// Mitsubishi GX Works2 project: PLC_GROUP18   PLC: FX3G
// פרויקט אוטומציה

// global labels: Global1
VAR_GLOBAL
  StartWorkingDay AT X007 : BOOL;
  EmergencyButton AT X005 : BOOL;
  WorkingDay AT Y007 : BOOL;
  InputChocolate AT D1101 : REAL;
  InputNuts AT D1103 : REAL;
  InputPistacho AT D1105 : REAL;
  InputKadaif AT D1107 : REAL;
  M_20 AT M20 : BOOL;
END_VAR
VAR_GLOBAL CONSTANT
  MinChocolate : REAL := 400.0;
  MinNuts : REAL := 100.0;
  MinPistacho : REAL := 120.0;
  MinKadaif : REAL := 60.0;
END_VAR
VAR_GLOBAL
  StockChocolate AT D1109 : REAL;
  StockNuts AT D1111 : REAL;
  StockPistacho AT D1113 : REAL;
  StockKadaif AT D1115 : REAL;
  M_21 AT M21 : BOOL;
  StartMelt AT X001 : BOOL;
  MeltContainer AT D1117 : REAL;
END_VAR
VAR_GLOBAL CONSTANT
  Choco_400 : REAL := 400.0;
END_VAR
VAR_GLOBAL
  MeltProcess AT Y001 : BOOL;
  CastingTime AT TC1 : BOOL;
END_VAR
VAR_GLOBAL CONSTANT
  DoneMelt : INT := 45;
END_VAR
VAR_GLOBAL
  FinishCasting AT TS1 : BOOL;
  SampleType AT X004 : BOOL;
  AnalogInput1 AT D8280 : INT;
  FloatInput1 AT D1119 : REAL;
  M_22 AT M22 : BOOL;
  M_23 AT M23 : BOOL;
  M_24 AT M24 : BOOL;
  M_25 AT M25 : BOOL;
END_VAR
VAR_GLOBAL CONSTANT
  Div400 : REAL := 400;
  Cons5 : REAL := 5.0;
END_VAR
VAR_GLOBAL
  MixNuts AT M26 : BOOL;
  DubalChoco AT M27 : BOOL;
END_VAR
VAR_GLOBAL CONSTANT
  Nuts100 : REAL := 100;
  Pistacho100 : REAL := 100;
END_VAR
VAR_GLOBAL
  FillContainer AT D1121 : REAL;
END_VAR
VAR_GLOBAL CONSTANT
  Amount200 : REAL := 200;
END_VAR
VAR_GLOBAL
  Sen_temp AT X002 : BOOL;
  EmplyTemplates AT X003 : BOOL;
END_VAR
VAR_GLOBAL CONSTANT
  Casting4sec : INT := 40;
END_VAR
VAR_GLOBAL
  CastingProcess AT Y002 : BOOL;
END_VAR
VAR_GLOBAL CONSTANT
  Nuts20 : REAL := 20;
  Pistacho120 : REAL := 120;
  Kadaif60 : REAL := 60;
END_VAR
VAR_GLOBAL
  Y_3 AT Y003 : BOOL;
  Y_4 AT Y004 : BOOL;
  TC_3 AT TC3 : BOOL;
END_VAR
VAR_GLOBAL CONSTANT
  FlashTime : INT := 10;
END_VAR
VAR_GLOBAL
  TS_3 AT TS3 : BOOL;
  TC_4 AT TC4 : BOOL;
  TS_4 AT TS4 : BOOL;
  Cooling AT X006 : BOOL;
END_VAR
VAR_GLOBAL CONSTANT
  Flash5 : INT := 50;
END_VAR
VAR_GLOBAL
  TC_2 AT TC2 : BOOL;
  TS_2 AT TS2 : BOOL;
  CoolContainer AT D1123 : REAL;
END_VAR
VAR_GLOBAL CONSTANT
  Cool3 : INT := 30;
END_VAR
VAR_GLOBAL
  CoolTime AT TC6 : BOOL;
  TS_6 AT TS6 : BOOL;
  CoolingProcess AT Y006 : BOOL;
  CastingContainer AT D1125 : REAL;
END_VAR
VAR_GLOBAL CONSTANT
  Reset : REAL;
END_VAR
VAR_GLOBAL
  M_28 AT M28 : BOOL;
  M_29 AT M29 : BOOL;
  X_0 AT X000 : BOOL;
  Y_5 AT Y005 : BOOL;
  FirstC AT CC1 : BOOL;
  OutC1 AT CS1 : BOOL;
END_VAR
VAR_GLOBAL CONSTANT
  CounterThreeTimes : WORD := 4;
END_VAR
VAR_GLOBAL
  FinishPacking AT M51 : BOOL;
  PacksContainer AT D1127 : REAL;
END_VAR
VAR_GLOBAL CONSTANT
  AddPack : REAL := 1;
END_VAR
VAR_GLOBAL
  M_52 AT M52 : BOOL;
  M_53 AT M53 : BOOL;
  M_60 AT M60 : BOOL;
  Packages AT D1129 : REAL;
  Analog_output AT D8282 : INT;
END_VAR
VAR_GLOBAL CONSTANT
  Cons40 : REAL := 40.0;
  ResetWord : INT;
END_VAR
VAR_GLOBAL
  X_10 AT X010 : BOOL;
  M_30 AT M30 : BOOL;
  M_31 AT M31 : BOOL;
END_VAR

// task Task_01 (event TRUE, interval 0, priority 31): POU_01

PROGRAM POU_01
(* structured ladder/FBD written out as ST: instructions are called as NAME(EN, inputs, outputs); _pN, _eN, _tN stand for wires *)
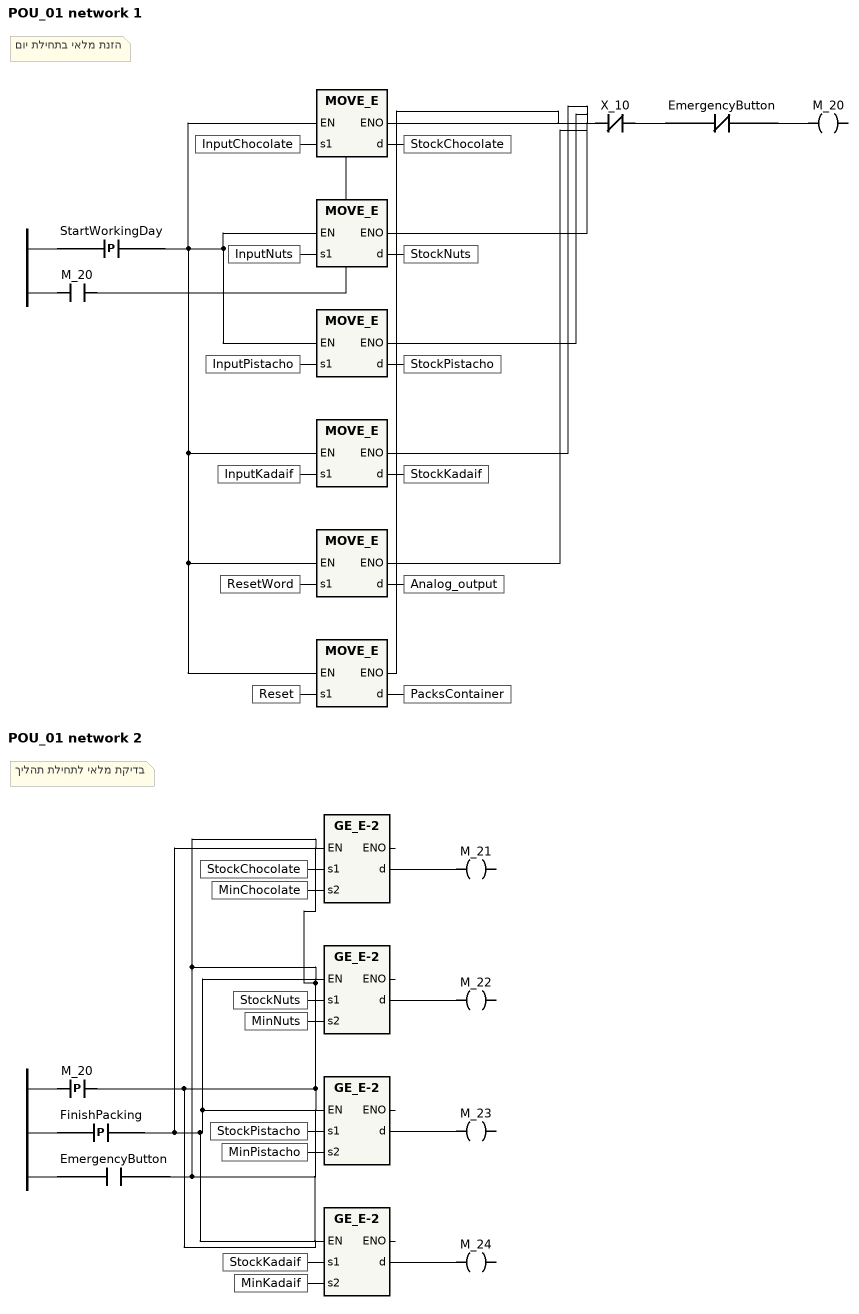
(* network 1 *)
(* הזנת מלאי בתחילת יום *)
_p1 := LDP(TRUE, StartWorkingDay);
_e2 := MOVE_E(_p1, InputChocolate, StockChocolate);
_e3 := MOVE_E(_p1, InputNuts, StockNuts);
_e4 := MOVE_E(_p1, InputPistacho, StockPistacho);
_e5 := MOVE_E(_p1, InputKadaif, StockKadaif);
_e6 := MOVE_E(_p1, ResetWord, Analog_output);
_e7 := MOVE_E(_p1, Reset, PacksContainer);
M_20 := ((_e2 OR _e3 OR _e4 OR _e5 OR _e6 OR _e7 OR M_20) AND NOT X_10) AND NOT EmergencyButton;
(* network 2 *)
(* בדיקת מלאי לתחילת תהליך *)
_p1 := LDP(TRUE, M_20) OR LDP(TRUE, FinishPacking) OR EmergencyButton;
GE_E(_p1, StockChocolate, MinChocolate, _t2);
M_21 := _t2;
GE_E(_p1, StockNuts, MinNuts, _t3);
M_22 := _t3;
GE_E(_p1, StockPistacho, MinPistacho, _t4);
M_23 := _t4;
GE_E(_p1, StockKadaif, MinKadaif, _t5);
M_24 := _t5;
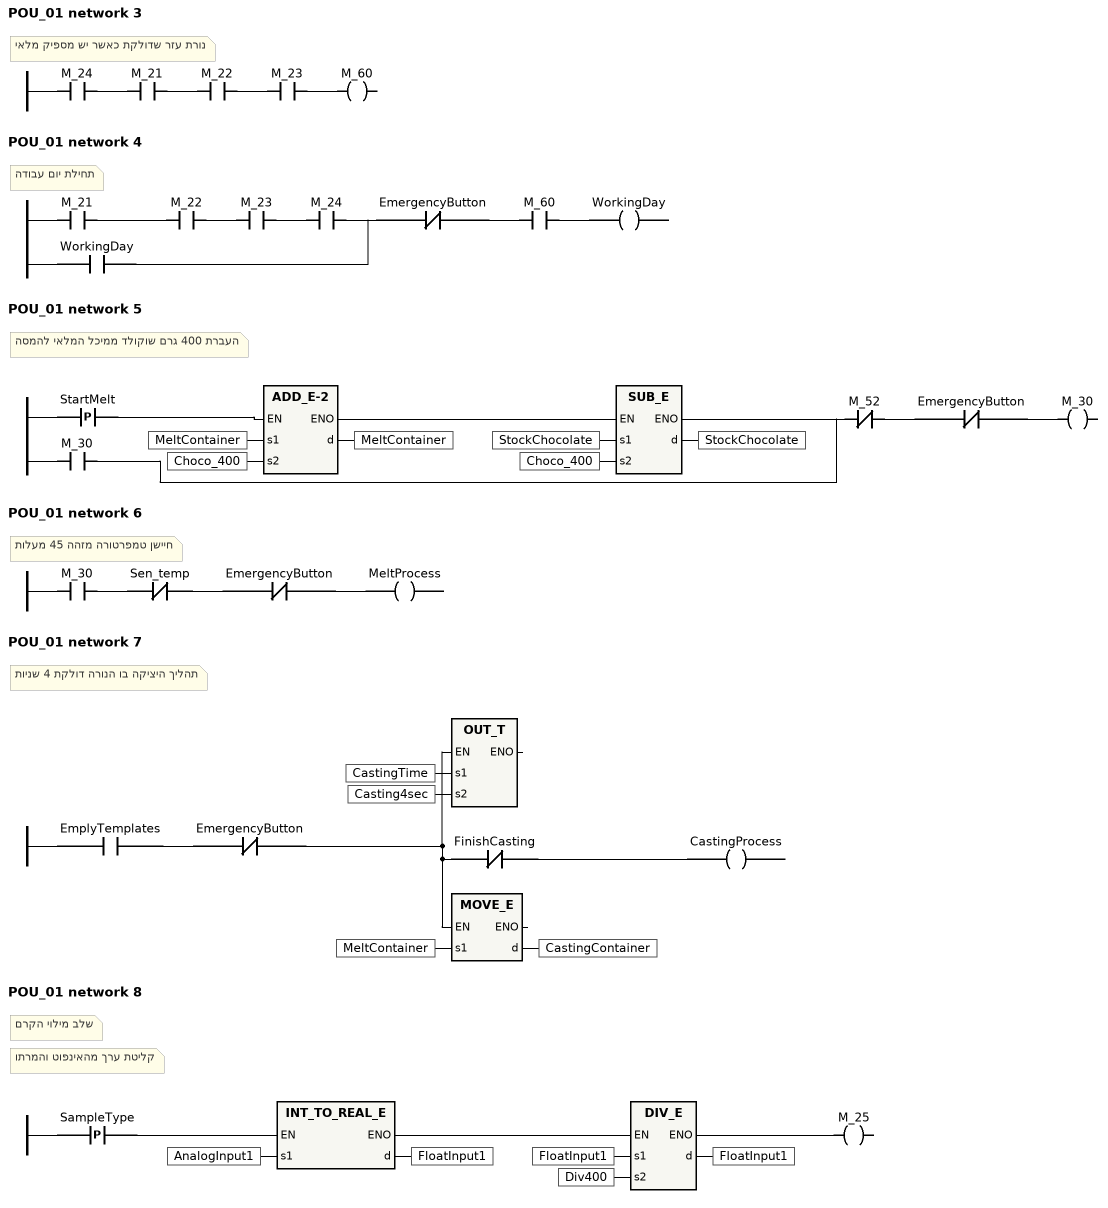
(* network 3 *)
(* נורת עזר שדולקת כאשר יש מספיק מלאי *)
M_60 := M_24 AND M_21 AND M_22 AND M_23;
(* network 4 *)
(* תחילת יום עבודה *)
WorkingDay := (((M_21 AND M_22 AND M_23 AND M_24) OR WorkingDay) AND NOT EmergencyButton) AND M_60;
(* network 5 *)
(* העברת 400 גרם שוקולד ממיכל המלאי להמסה *)
_e1 := ADD_E(LDP(TRUE, StartMelt), MeltContainer, Choco_400, MeltContainer);
_e2 := SUB_E(_e1, StockChocolate, Choco_400, StockChocolate);
M_30 := ((_e2 OR M_30) AND NOT M_52) AND NOT EmergencyButton;
(* network 6 *)
(* חיישן טמפרטורה מזהה 45 מעלות *)
MeltProcess := M_30 AND NOT Sen_temp AND NOT EmergencyButton;
(* network 7 *)
(* תהליך היציקה בו הנורה דולקת 4 שניות *)
_p1 := EmplyTemplates AND NOT EmergencyButton;
OUT_T(_p1, CastingTime, Casting4sec);
CastingProcess := _p1 AND NOT FinishCasting;
MOVE_E(_p1, MeltContainer, CastingContainer);
(* network 8 *)
(* שלב מילוי הקרם *)
(* קליטת ערך מהאינפוט והמרתו *)
_e1 := INT_TO_REAL_E(LDP(TRUE, SampleType), AnalogInput1, FloatInput1);
_e2 := DIV_E(_e1, FloatInput1, Div400, FloatInput1);
M_25 := _e2;
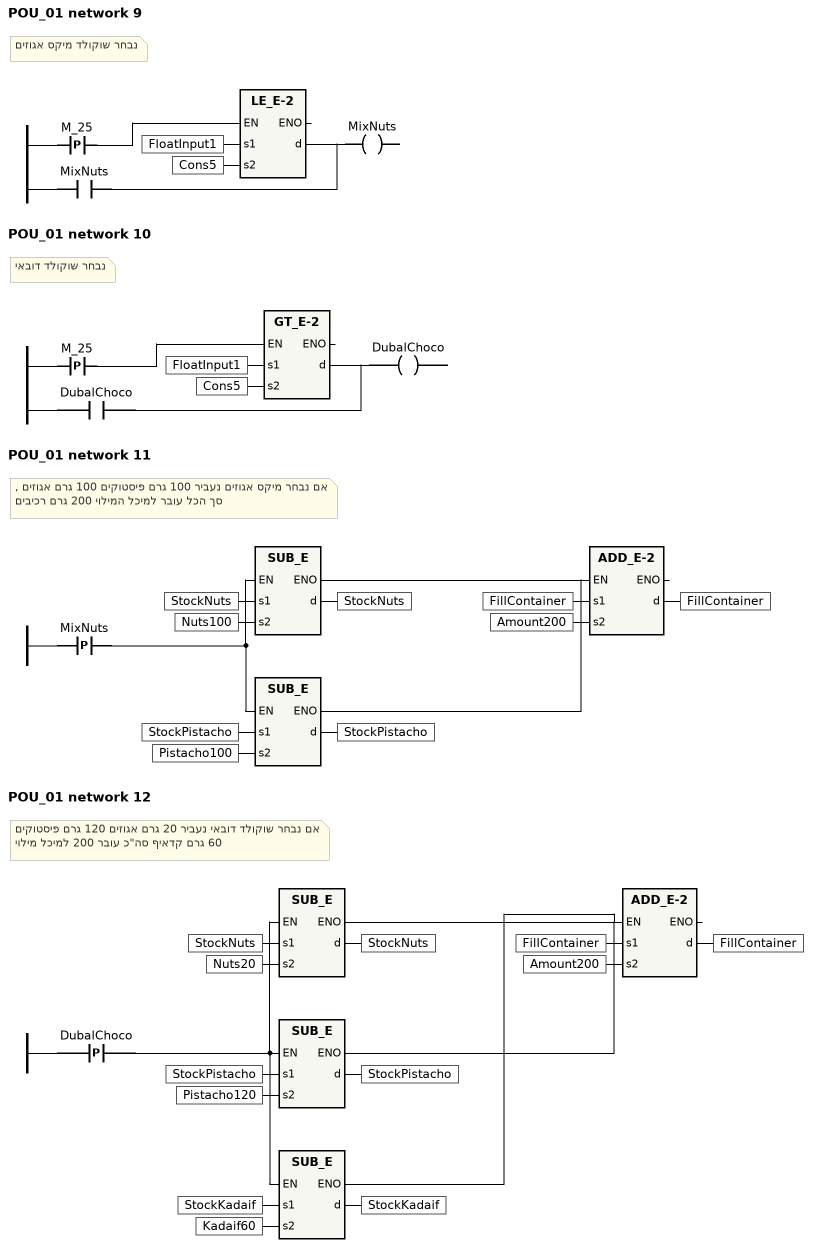
(* network 9 *)
(* נבחר שוקולד מיקס אגוזים *)
LE_E(LDP(TRUE, M_25), FloatInput1, Cons5, _t1);
MixNuts := _t1 OR MixNuts;
(* network 10 *)
(* נבחר שוקולד דובאי *)
GT_E(LDP(TRUE, M_25), FloatInput1, Cons5, _t1);
DubalChoco := _t1 OR DubalChoco;
(* network 11 *)
(* אם נבחר מיקס אגוזים נעביר 100 גרם פיסטוקים 100 גרם אגוזים , סך הכל עובר למיכל המילוי 200 גרם רכיבים *)
_p1 := LDP(TRUE, MixNuts);
_e2 := SUB_E(_p1, StockNuts, Nuts100, StockNuts);
_e3 := SUB_E(_p1, StockPistacho, Pistacho100, StockPistacho);
ADD_E(_e2 OR _e3, FillContainer, Amount200, FillContainer);
(* network 12 *)
(* אם נבחר שוקולד דובאי נעביר 20 גרם אגוזים 120 גרם פיסטוקים 60 גרם קדאיף סה"כ עובר 200 למיכל מילוי *)
_p1 := LDP(TRUE, DubalChoco);
_e2 := SUB_E(_p1, StockNuts, Nuts20, StockNuts);
_e3 := SUB_E(_p1, StockPistacho, Pistacho120, StockPistacho);
_e4 := SUB_E(_p1, StockKadaif, Kadaif60, StockKadaif);
ADD_E(_e2 OR _e3 OR _e4, FillContainer, Amount200, FillContainer);
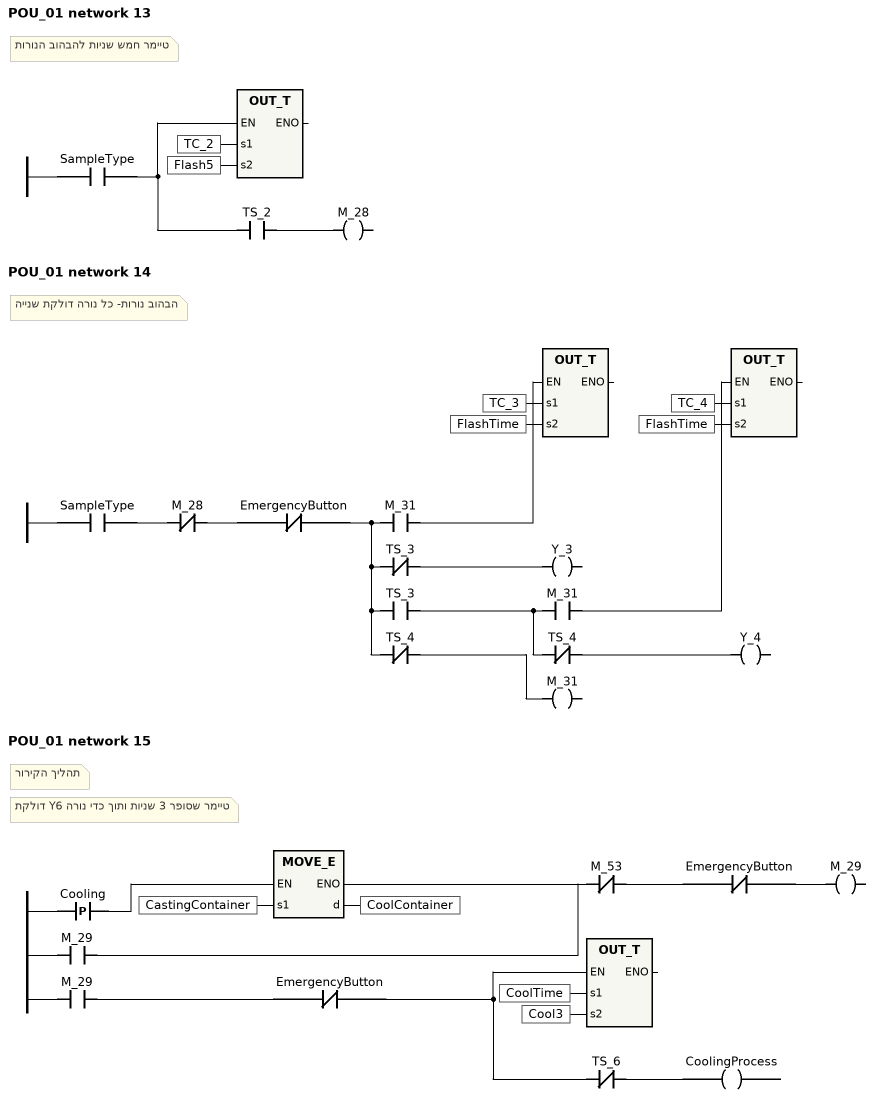
(* network 13 *)
(* טיימר חמש שניות להבהוב הנורות *)
OUT_T(SampleType, TC_2, Flash5);
M_28 := SampleType AND TS_2;
(* network 14 *)
(* הבהוב נורות- כל נורה דולקת שנייה *)
_p1 := SampleType AND NOT M_28 AND NOT EmergencyButton;
OUT_T(_p1 AND M_31, TC_3, FlashTime);
Y_3 := _p1 AND NOT TS_3;
_p2 := _p1 AND TS_3;
OUT_T(_p2 AND M_31, TC_4, FlashTime);
Y_4 := _p2 AND NOT TS_4;
M_31 := _p1 AND NOT TS_4;
(* network 15 *)
(* תהליך הקירור *)
(* טיימר שסופר 3 שניות ותוך כדי נורה Y6 דולקת *)
_e1 := MOVE_E(LDP(TRUE, Cooling), CastingContainer, CoolContainer);
M_29 := ((_e1 OR M_29) AND NOT M_53) AND NOT EmergencyButton;
_p2 := M_29 AND NOT EmergencyButton;
OUT_T(_p2, CoolTime, Cool3);
CoolingProcess := _p2 AND NOT TS_6;
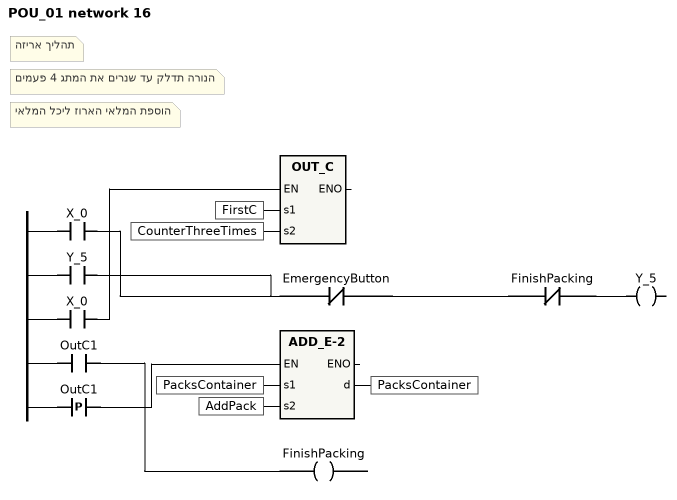
(* network 16 *)
(* תהליך אריזה *)
(* הנורה תדלק עד שנרים את המתג 4 פעמים *)
(* הוספת המלאי הארוז ליכל המלאי *)
Y_5 := ((X_0 OR Y_5) AND NOT EmergencyButton) AND NOT FinishPacking;
OUT_C(X_0, FirstC, CounterThreeTimes);
FinishPacking := OutC1;
ADD_E(LDP(TRUE, OutC1), PacksContainer, AddPack, PacksContainer);
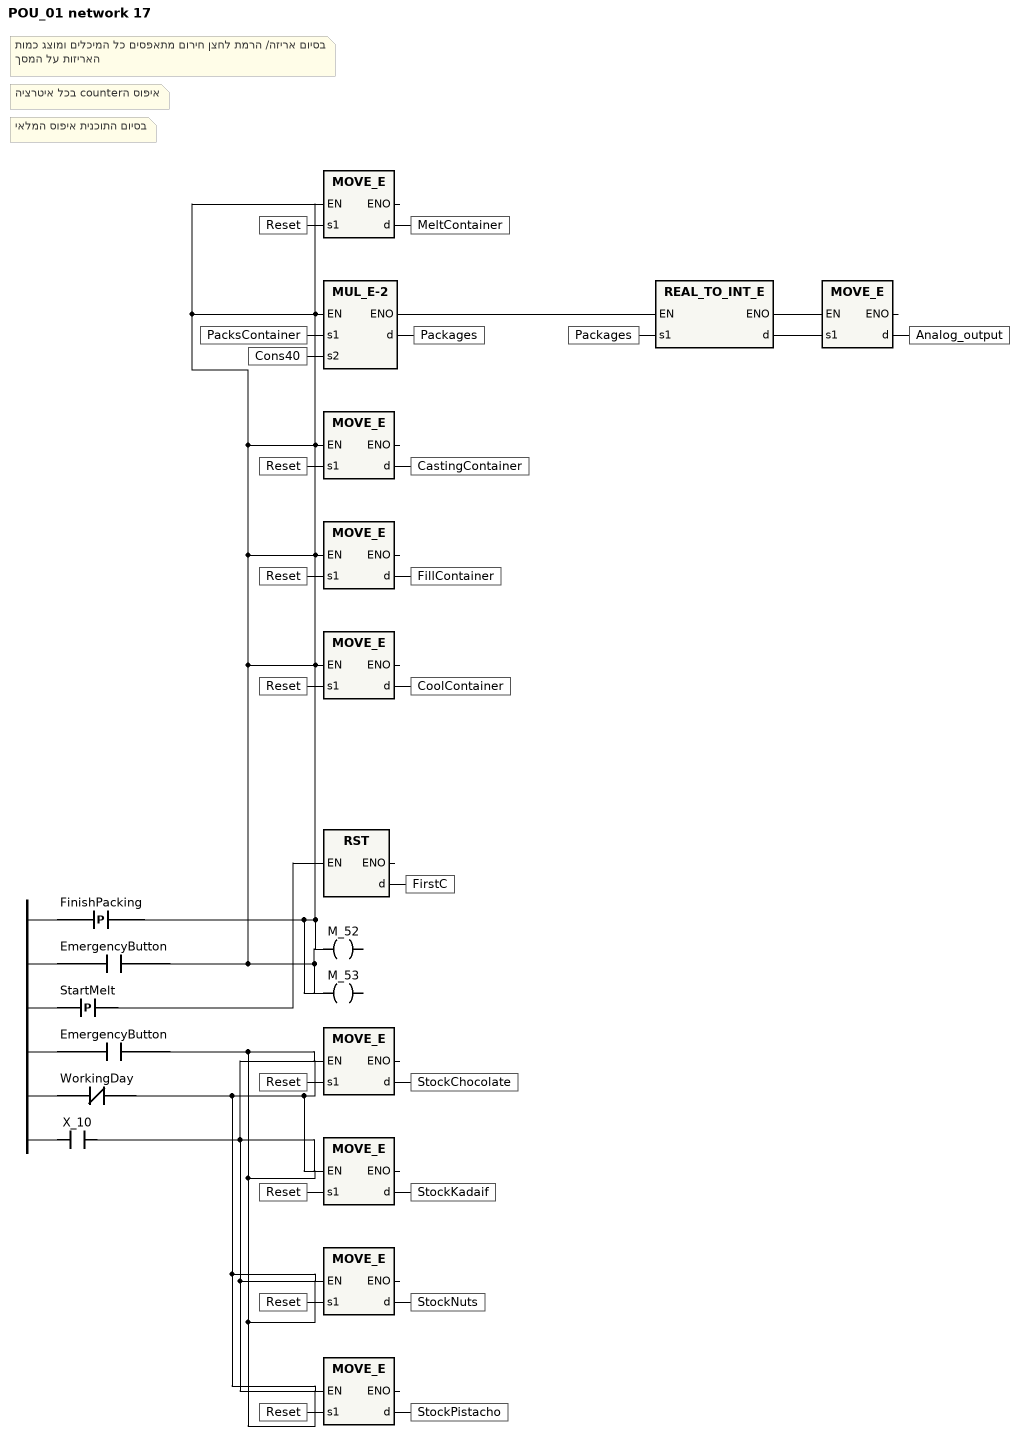
(* network 17 *)
(* בסיום אריזה/ הרמת לחצן חירום מתאפסים כל המיכלים ומוצג כמות האריזות על המסך *)
(* איפוס הcounter בכל איטרציה *)
(* בסיום התוכנית איפוס המלאי *)
_p1 := LDP(TRUE, FinishPacking) OR EmergencyButton;
MOVE_E(_p1, Reset, MeltContainer);
MOVE_E(_p1, Reset, CastingContainer);
MOVE_E(_p1, Reset, FillContainer);
MOVE_E(_p1, Reset, CoolContainer);
M_52 := _p1;
M_53 := _p1;
_e2 := MUL_E(_p1, PacksContainer, Cons40, Packages);
_e4 := REAL_TO_INT_E(_e2, Packages, _t3);
MOVE_E(_e4, _t3, Analog_output);
RST(LDP(TRUE, StartMelt), FirstC);
_p5 := EmergencyButton OR (NOT WorkingDay) OR X_10;
MOVE_E(_p5, Reset, StockChocolate);
MOVE_E(_p5, Reset, StockKadaif);
MOVE_E(_p5, Reset, StockNuts);
MOVE_E(_p5, Reset, StockPistacho);
END_PROGRAM
